Fanuc TP program (LS listing): Pick_Entrada.ls

/PROG  Pick_Entrada
/ATTR
OWNER       = MNEDITOR;
COMMENT     = ""
PROG_SIZE   = 913;
CREATE      = DATE 23-04-22  TIME 19:45:13;
MODIFIED      = DATE 23-04-22  TIME 19:45:13;
FILE_NAME   = ;
VERSION    = 0;
LINE_COUNT  = 13;
MEMORY_SIZE = 1197;
PROTECT     = READ_WRITE;
TCD:  STACK_SIZE    = 0,
      TASK_PRIORITY = 50,
      TIME_SLICE    = 0,
      BUSY_LAMP_OFF = 0,
      ABORT_REQUEST = 0,
      PAUSE_REQUEST = 0;
DEFAULT_GROUP   = 1,*,*,*,*,*,*,* ;
CONTROL_CODE    = 00000000 00000000;
/APPL
/MN
1:!FANUC America Corp. ;
2:!ROBOGUIDE Generated This TPP ;
3:!Run SimPRO.cf to setup frame and tool data ;
4:!This program will be overwritten on the next save or run. ;
5:! Pickup ('Parte Soldadura') From ('Conveyorn Entrada:Link1') With ('GP: 1 - UT: 1  (TCP_Gripper)') ;
7:!WAIT 0.00 (sec) ;
/POS
/END
